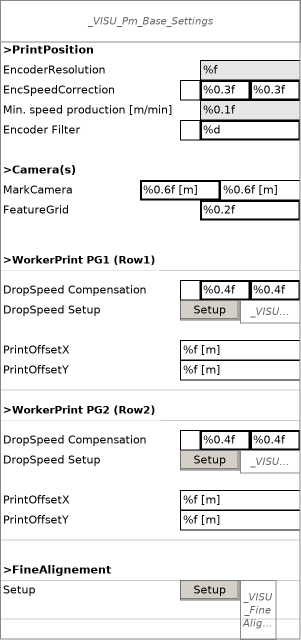
VISUALIZATION _VISU_Pm_WEU_Settings  // 301x640
VAR_IN_OUT
	mInst : FB_PrintModule_WEU;
END_VAR
    Rectangle (0,580 300x39)
    Rectangle (250,80 50x20), "%0.3f", tooltip "Encoder speed compensation reference speed", text variable: mInst.fbPrintPosition._fSpeedCompRefSpeed
        OnMouseClick: write the text variable via Default
    Rectangle (200,80 50x20), "%0.3f", tooltip "Encoder speed compensation factor", text variable: mInst.fbPrintPosition._fSpeedCompFactor
        OnMouseClick: write the text variable via Default
    RoundedRectangle (180,80 20x20)
        toggle mInst.fbPrintPosition._bEnSpeedComp
    Rectangle (0,80 180x20), "EncSpeedCorrection"
    Rectangle (0,60 180x20), "EncoderResolution"
    Rectangle (200,60 100x20), "%f", tooltip "by calculation", text variable: mInst.fbPrintPosition._fEncoderResolution
    Rectangle (0,270 300x120)
    Rectangle (0,280 180x20), "DropSpeed Compensation"
    Rectangle (200,280 50x20), "%0.4f", tooltip "DropSpeed [m/s]", text variable: mInst.fbWorkerPrint[1].fbDropSpeedComp.fDropSpeed
        OnMouseClick: write the text variable via Default
    Rectangle (250,280 50x20), "%0.4f", tooltip "Dead/Add Time [ms]", text variable: mInst.fbWorkerPrint[1].fbDropSpeedComp.fDropSpeedDeadTime
        OnMouseClick: write the text variable via Default
    RoundedRectangle (180,280 20x20), tooltip "Enabled compensation", input disabled if: TRUE
        toggle mInst.fbWorkerPrint[1].fbDropSpeedComp._bEnable p2164770859=TRUE
    Button (180,300 60x20), "Setup", tooltip "Setup"
        toggle mInst.fbWorkerPrint[1].bShowDropSpeedSetup
    Rectangle (0,300 180x20), "DropSpeed Setup"
    Rectangle (0,40 180x20), ">PrintPosition"
    Rectangle (0,100 180x20), "Min. speed production [m/min]"
    Rectangle (200,100 100x20), "%0.1f", tooltip "constant", text variable: mInst.fC_ProductionSpeedMpMin_Level
    Rectangle (0,160 180x20), ">Camera(s)"
    Rectangle (220,180 80x20), "%0.6f [m]", tooltip "(not used) CameraToPrintUnit", text variable: mInst.fbMarkCameraWeu._fCameraToPrintOffset, input disabled if: TRUE
        OnMouseDown: write the text variable via Default
    Rectangle (140,180 80x20), "%0.6f [m]", tooltip "DetectToCamera", text variable: mInst.fbMarkCameraWeu._fDetectToCameraOffset
        OnMouseDown: write the text variable via Default
    Rectangle (0,180 140x20), "MarkCamera"
    Rectangle (200,120 100x20), "%d", tooltip "Filter depth", text variable: mInst.fbPrintPosition.fbPositionMaster.nFilterDepth
        OnMouseClick: write the text variable via Default
    RoundedRectangle (180,120 20x20)
        toggle mInst.fbPrintPosition.fbPositionMaster.bEnableFilter
    Rectangle (0,120 180x20), "Encoder Filter"
    Rectangle (0,200 180x20), "FeatureGrid"
    Rectangle (200,200 100x20), "%0.2f", text variable: mInst.fbWorkerCamera._fFeatureGrid
        OnMouseDown: write the text variable via Default
    Rectangle (0,560 180x20), ">FineAlignement"
    Button (180,580 60x20), "Setup", tooltip "Setup"
        toggle minst.fbView.bShowFineAlignement
    Rectangle (0,580 180x20), "Setup"
    Frame (0,0 301x42)
        shows _VISU_Pm_Base_Settings(mInst := mInst)
    Rectangle (0,340 180x20), "PrintOffsetX"
    Rectangle (0,360 180x20), "PrintOffsetY"
    Rectangle (180,340 120x20), "%f [m]", text variable: mInst.fbWorkerPrint[1].fPrintStartOffset, input disabled if: TRUE
    Rectangle (180,360 120x20), "%f [m]", text variable: mInst.fbWorkerPrint[1].fPrintYOffset, input disabled if: TRUE
    Frame (240,580 36x60), invisible if: NOT minst.fbView.bShowFineAlignement
        shows _VISU_FineAlignment(mInst := mInst.fbFineAlignement)
    Rectangle (0,420 300x120)
    Rectangle (0,430 180x20), "DropSpeed Compensation"
    Rectangle (200,430 50x20), "%0.4f", tooltip "DropSpeed [m/s]", text variable: mInst.fbWorkerPrint[2].fbDropSpeedComp.fDropSpeed
        OnMouseClick: write the text variable via Default
    Rectangle (250,430 50x20), "%0.4f", tooltip "Dead/Add Time [ms]", text variable: mInst.fbWorkerPrint[2].fbDropSpeedComp.fDropSpeedDeadTime
        OnMouseClick: write the text variable via Default
    RoundedRectangle (180,430 20x20), tooltip "Enabled compensation", input disabled if: TRUE
        toggle mInst.fbWorkerPrint[2].fbDropSpeedComp._bEnable p2164770859=TRUE
    Button (180,450 60x20), "Setup", tooltip "Setup"
        toggle mInst.fbWorkerPrint[2].bShowDropSpeedSetup
    Rectangle (0,450 180x20), "DropSpeed Setup"
    Rectangle (0,490 180x20), "PrintOffsetX"
    Rectangle (0,510 180x20), "PrintOffsetY"
    Rectangle (180,490 120x20), "%f [m]", text variable: mInst.fbWorkerPrint[2].fPrintStartOffset, input disabled if: TRUE
    Rectangle (180,510 120x20), "%f [m]", text variable: mInst.fbWorkerPrint[2].fPrintYOffset, input disabled if: TRUE
    Frame (240,450 60x23), invisible if: NOT mInst.fbWorkerPrint[2].bShowDropSpeedSetup
        shows _VISU_DropSpeedComp_Setup(mInst := mInst.fbWorkerPrint[2].fbDropSpeedComp)
    Rectangle (0,400 160x20), ">WorkerPrint PG2 (Row2)"
    Rectangle (0,250 160x20), ">WorkerPrint PG1 (Row1)"
    Frame (240,300 60x23), invisible if: NOT mInst.fbWorkerPrint[1].bShowDropSpeedSetup
        shows _VISU_DropSpeedComp_Setup(mInst := mInst.fbWorkerPrint[1].fbDropSpeedComp)
END_VISUALIZATION

(* stored: Version 1.1.0.1, ProductVersion 3.1.4024.11
   Visu _VISU_Pm_WEU_Settings: Id {42128b7e-6368-4298-b80c-e6d6bdbb0477} *)
